TYPE StepLog_Struct :
STRUCT
	step_number : DINT;
	created_at : LINT;
	program_name : STRING(80);
END_STRUCT
END_TYPE

(* stored: Version 1.1.0.1, ProductVersion 3.1.4026.13
   DUT StepLog_Struct: Id {14eba6f7-6a08-4ce8-88ac-e811c7521b85} *)
